TYPE ST_MatrixConfigs :
STRUCT
	InletConfig: ARRAY [1..GVL_HMI.cMaxRows,1..GVL_HMI.cMaxCols] OF ST_SolenoidConfig;
	FillConfig: ARRAY [1..GVL_HMI.cMaxRows,1..GVL_HMI.cMaxCols] OF ST_SolenoidConfig;
	DispenseConfig: ARRAY [1..GVL_HMI.cMaxRows,1..GVL_HMI.cMaxCols] OF ST_SolenoidConfig;
END_STRUCT
END_TYPE

(* stored: Version 1.1.0.1
   DUT ST_MatrixConfigs: Id {f1aa3f99-6346-4bcc-aef4-8b157aa6144e} *)
